FUNCTION_BLOCK PUSHER_MDL (* Pusher Model *)
  (* Standard: 61499-2 *)
  (* Version 0.2, 2003-12-05, JHC, Rockwell Automation, Renamed from NEWCOMPFB. *)
  (* Version 0.1, 2002-01-08, JHC, Rockwell Automation, Added DLY FB as example. *)
  (* Version 0.0, 2000-05-27, JHC, Rockwell Automation *)
  (* Compiler header: package fb.rt.dasdA1.A2; *)
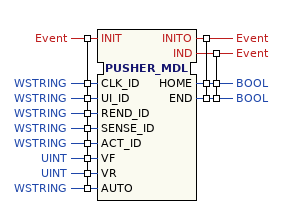
  EVENT_INPUT
    INIT WITH CLK_ID, UI_ID, REND_ID, SENSE_ID, ACT_ID, VF, VR, AUTO; (* Initialization Request *)
  END_EVENT
  EVENT_OUTPUT
    INITO WITH HOME, END; (* Initialization Confirm *)
    IND WITH HOME, END;
  END_EVENT
  VAR_INPUT
    CLK_ID : WSTRING;
    UI_ID : WSTRING;
    REND_ID : WSTRING;
    SENSE_ID : WSTRING;
    ACT_ID : WSTRING;
    VF : UINT;
    VR : UINT;
    AUTO : WSTRING; (* AUTO_ID *)
  END_VAR
  VAR_OUTPUT
    HOME : BOOL;
    END : BOOL;
  END_VAR
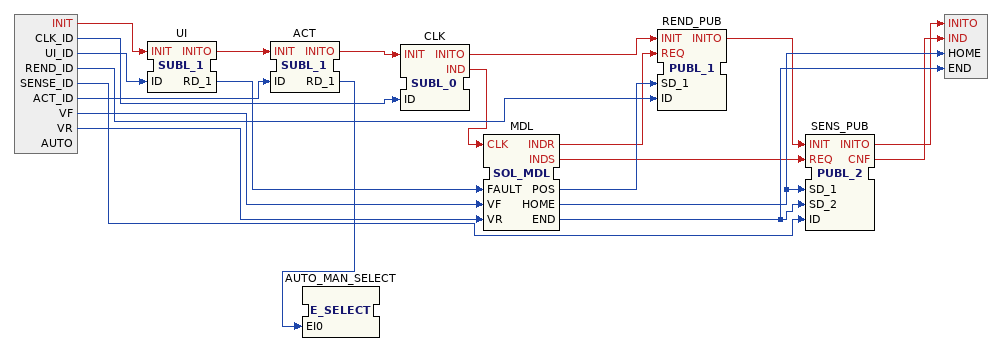
  FBS
    SENS_PUB : PUBL_2;
    MDL : SOL_MDL;
    REND_PUB : PUBL_1;
    CLK : SUBL_0;
    ACT : SUBL_1;
    UI : SUBL_1;
    AUTO_MAN_SELECT : E_SELECT;
  END_FBS
  EVENT_CONNECTIONS
    INIT TO UI.INIT;
    UI.INITO TO ACT.INIT;
    ACT.INITO TO CLK.INIT;
    CLK.INITO TO REND_PUB.INIT;
    REND_PUB.INITO TO SENS_PUB.INIT;
    MDL.INDR TO REND_PUB.REQ;
    MDL.INDS TO SENS_PUB.REQ;
    CLK.IND TO MDL.CLK;
    SENS_PUB.INITO TO INITO;
    SENS_PUB.CNF TO IND;
  END_CONNECTIONS
  DATA_CONNECTIONS
    MDL.POS TO REND_PUB.SD_1;
    MDL.HOME TO HOME;
    MDL.END TO END;
    MDL.HOME TO SENS_PUB.SD_1;
    MDL.END TO SENS_PUB.SD_2;
    UI.RD_1 TO MDL.FAULT;
    UI_ID TO UI.ID;
    ACT_ID TO ACT.ID;
    CLK_ID TO CLK.ID;
    REND_ID TO REND_PUB.ID;
    SENSE_ID TO SENS_PUB.ID;
    VF TO MDL.VF;
    VR TO MDL.VR;
    ACT.RD_1 TO AUTO_MAN_SELECT.EI0;
    ACT.RD_1 TO AUTO_MAN_SELECT.EI0;
  END_CONNECTIONS
END_FUNCTION_BLOCK
